// TIA Portal V18 export
TYPE "PLCtoMES_MainCheckOut_ext"
// stored: IsFailsafeCompliant false
   STRUCT
      Unload_Station1DataSaveReq : Bool;   // 本站工位1过程数据保存触发位
      Unload_Station2DataSaveReq : Bool;   // 本站工位2过程数据保存触发位
      Unload_Station3DataSaveReq : Bool;   // Spare
      Unload_Station4DataSaveReq : Bool;   // Spare
      Unload_Station5DataSaveReq : Bool;   // Spare
      Unload_Station6DataSaveReq : Bool;   // Spare
      Unload_Station7DataSaveReq : Bool;   // Spare
      Unload_Station8DataSaveReq : Bool;   // Spare
   END_STRUCT;
END_TYPE
